INTERFACE I_MotionDrive

END_INTERFACE

(* stored: Version 1.1.0.1
   Itf I_MotionDrive: Id {848572bc-fef8-4708-bb80-0dc37710e2cf} *)
